FUNCTION_BLOCK PAEActFlap EXTENDS PAEActuator1way
VAR_INPUT
END_VAR
VAR_OUTPUT
END_VAR
VAR
END_VAR

END_FUNCTION_BLOCK

(* stored: Version 1.1.0.1, ProductVersion 3.1.4020.12
   POU PAEActFlap: Id {496459d0-1036-4764-ab4a-0abe57fdc608}, SpecialFunc None *)
